FUNCTION_BLOCK fb_oeprationPush
VAR_INPUT
END_VAR
VAR_OUTPUT
END_VAR
VAR
	SFCInit : bool;
	flgInitDone: BOOL;
	trn_chuckOpenDone: BOOL;
	trn_chuckCloseDone: BOOL;
	trn_gm_chuckOpenDone: BOOL;
	trn_gm_chuckCloseDone: BOOL;
END_VAR

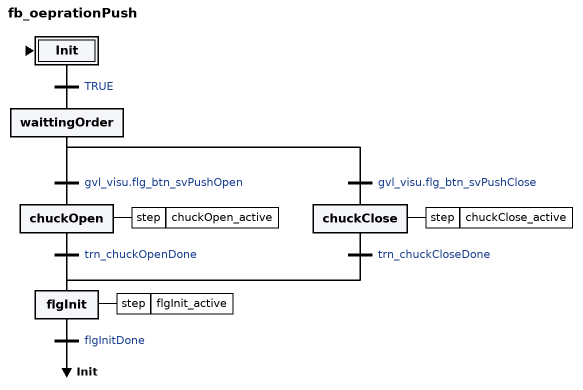
INITIAL_STEP Init:
END_STEP
TRANSITION FROM Init TO waittingOrder
    := TRUE;
END_TRANSITION
STEP waittingOrder:
END_STEP
TRANSITION FROM waittingOrder TO chuckOpen
    := gvl_visu.flg_btn_svPushOpen;
END_TRANSITION
STEP chuckOpen:
    chuckOpen_active(N);  // step action
END_STEP
TRANSITION FROM chuckOpen TO flgInit
    := trn_chuckOpenDone;
END_TRANSITION
TRANSITION FROM waittingOrder TO chuckClose
    := gvl_visu.flg_btn_svPushClose;
END_TRANSITION
STEP chuckClose:
    chuckClose_active(N);  // step action
END_STEP
TRANSITION FROM chuckClose TO flgInit
    := trn_chuckCloseDone;
END_TRANSITION
STEP flgInit:
    flgInit_active(N);  // step action
END_STEP
TRANSITION FROM flgInit TO Init
    := flgInitDone;
END_TRANSITION

ACTION chuckClose_active:
IF chuckClose._x AND chuckClose.x = FALSE THEN
	trn_chuckCloseDone := FALSE;
	gvl_solv.fbi_push.in_flg_run := FALSE;
	gvl_solv.fbi_push.in_var_moveMode := eP_svMoveMode.svB;
ELSIF chuckClose._x AND chuckClose.x THEN
	gvl_solv.fbi_push.in_flg_run := TRUE;
	IF gvl_solv.fbi_push.out_flg_Done THEN
		gvl_solv.fbi_push.in_flg_run := FALSE;
		trn_chuckCloseDone := TRUE;
	END_IF
END_IF
END_ACTION

ACTION chuckOpen_active:
IF chuckOpen._x AND chuckOpen.x = FALSE THEN
	trn_chuckOpenDone := FALSE;
	gvl_solv.fbi_push.in_flg_run := FALSE;
	gvl_solv.fbi_push.in_var_moveMode := eP_svMoveMode.svA;
ELSIF chuckOpen._x AND chuckOpen.x THEN
	gvl_solv.fbi_push.in_flg_run := TRUE;
	IF gvl_solv.fbi_push.out_flg_Done THEN
 		gvl_solv.fbi_push.in_flg_run := FALSE;
		trn_chuckOpenDone := TRUE;
	END_IF
END_IF
END_ACTION

ACTION flgInit_active:
IF flgInit._x AND flgInit.x = FALSE THEN
	flgInitDone := FALSE;
	gvl_visu.flg_btn_svPushOpen := FALSE;
	gvl_visu.flg_btn_svPushClose := FALSE;
ELSIF flgInit._x AND flgInit.x THEN
	flgInitDone := TRUE;
END_IF
END_ACTION

PROPERTY p_Init : bool
GET
p_init := THIS^.SFCInit;
END_GET
SET
THIS^.SFCInit := p_Init;
END_SET
END_PROPERTY

END_FUNCTION_BLOCK

(* stored: Version 1.1.0.1, ProductVersion 3.1.4024.11
   POU fb_oeprationPush: Id {69da8179-1ebb-4da3-8c77-c0ce35844780}, SpecialFunc None
   Action chuckClose_active: Id {bb6b388d-d3c1-498a-bb8d-b8afe911ff0a}
   Action chuckOpen_active: Id {0736c763-5e9c-4a7f-8d9e-e087c2956899}
   Action flgInit_active: Id {b6a3e1f2-e083-4202-98dd-ae59b0cbfc63}
   Property p_Init: Id {aca710df-c09f-43a7-a94f-e061c7a8de3a}
   Get Get: Id {fab33768-449c-4bc5-8c26-a281df06a949}
   Set Set: Id {aa733948-36ad-4dd2-ae87-707eb2aabbc8} *)
